Yaskawa INFORM job: LOAD_TOP_END_XYZ.JBI

/JOB
//NAME LOAD_TOP_END_XYZ
///FOLDERNAME FOLDER001
//POS
///NPOS 0,0,0,1,0,0
///TOOL 1
///POSTYPE ROBOT
///RECTAN
///RCONF 1,0,0,0,0,0,0,0,0,0,0,0,0,0,0,0,0,0,0,0,0,0,0,0
P00125=1116.664,160.780,493.887,-179.9993,-9.9981,-0.0025
//INST
///DATE 2025/09/29 14:33
///ATTR SC,RW
///GROUP1 RB1
NOP
'GET X Y Z VALUE FOR TOP END
'X
GETE D067 P125 (1)
SET I067  EXPRESS I066 * 100
IFTHENEXP I067>10000
	 SET I067 10000
ELSEIFEXP I067<-10000
	 SET I067 -10000
ENDIF
'Y
GETE D069 P125 (2)
SET I069  EXPRESS I068 * 100
IFTHENEXP I069>10000
	 SET I069 10000
ELSEIFEXP I069<-10000
	 SET I069 -10000
ENDIF
'Z
GETE D071 P125 (3)
SET I071  EXPRESS I070 * 100
IFTHENEXP I071>10000
	 SET I071 10000
ELSEIFEXP I071<-10000
	 SET I071 -10000
ENDIF
'ADD THE CORRECTIONS
ADD D067 I067
SETE P125 (1) D067
ADD D069 I069
SETE P125 (2) D069
ADD D071 I071
SETE P125 (3) D071
'SET TO 0
SET I066 0
SET I067 0
SET I068 0
SET I069 0
SET I070 0
SET I071 0
END
